Universal Robots PolyScope program: ccc_place_stick.urp

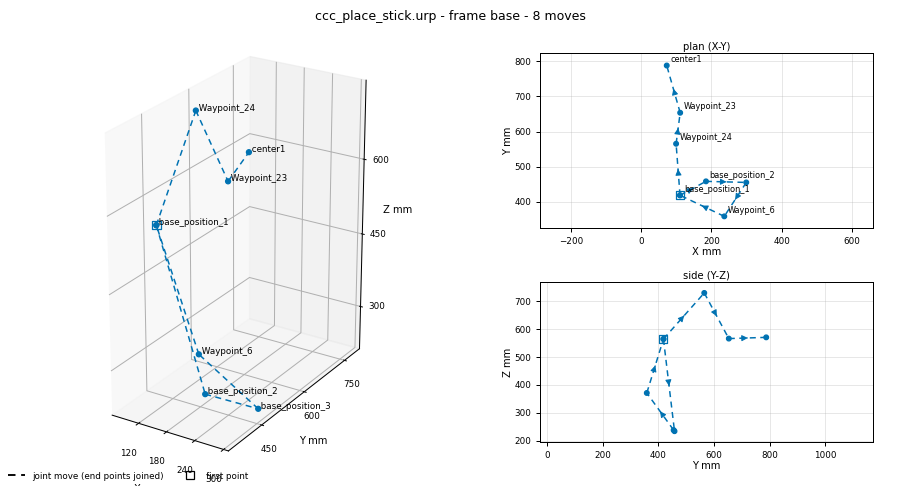
[picture p0: tool path of ccc_place_stick.urp in frame base, 8 of 8 moves have a stored position in this frame; points joined in program order, loops and branches not executed]
Program ccc_place_stick (installation=default directory=/programs/Nicolas_Arteaga/quality createdIn=5.12.4.1101661 lastSavedIn=5.12.4.1101661 robotSerialNumber=20225502378)
Calibrated DH parameters: a=[0.00022, -0.425328, -0.389701, 0.000059, 0.000065, 0]; d=[0.162608, 0.803456, 9.992211, -10.662202, 0.099702, 0.099559]; alpha=[1.570756, 0.001543, 0.004316, 1.570651, -1.570122, 0]; deltaTheta=[0, 0.002917, 0.116094, -0.119008, 0, -0.000001]
Robot Program (runOnlyOnce=true)
  'Takes the first wood stick and places it in the center of the cotton candy machine'
  MoveJ speed 60 deg/s, acceleration 80 deg/s^2 (useActiveTCP=true) feature=Base
    Waypoint base_position_1: TCP in base x=110.873 y=418.875 z=565.206 mm, rx=-1.5602 ry=-0.9891 rz=-1.3624 rad; joints [200.91, -129.117, 99.415, 36.172, 41.428, 90] deg; TCP offset x=0 y=0 z=191.5 mm, rx=0 ry=0 rz=0 rad
    Waypoint base_position_2: TCP in base x=184.715 y=458.614 z=234.006 mm, rx=-1.6866 ry=-0.757 rz=-1.7388 rad; joints [238.232, -104.263, 143.888, -41.533, 99.714, 90.08] deg; TCP offset x=0 y=0 z=191.5 mm, rx=0 ry=0 rz=0 rad
    URCap Gripper Activate (Robotiq_Grippers, Robotiq Inc.) dataModel(ResetAndActivateKey=false)
    URCap Gripper (Robotiq_Grippers, Robotiq Inc.) dataModel(forceInDouble=100.0, speedInDouble=100.0, position=78.0, force=100.0, speed=100.0, positionInDouble=78.0, slaveIds=[9], blocking=true)
    Waypoint base_position_3: TCP in base x=299.306 y=455.502 z=237.992 mm, rx=0.0242 ry=1.587 rz=-0.0069 rad; joints [252.253, -72.527, 107.61, -31.252, 163.421, 274.35] deg; TCP offset x=0 y=0 z=191.5 mm, rx=0 ry=0 rz=0 rad
    stick := GP_int_in[4]
    SuppressedNode
      stick := 10
    Loop While (checkContinuously=false) expression=stick>0
      MoveL speed 250 mm/s, acceleration 1200 mm/s^2 (useActiveTCP=true) feature=Base
        MoveDirectionNode (selectedDirection=ZMinus)
          Until DISTANCE (allowActions=false deceleration=3 distanceNodeType=STOP) Distance=0.016; motionParameters(blendRadius=0)
      stick := stick-1
    MoveL speed 250 mm/s, acceleration 1200 mm/s^2 (useActiveTCP=true) feature=Base
      MoveDirectionNode (selectedDirection=XPlus)
        Until DISTANCE (allowActions=false deceleration=3 distanceNodeType=STOP) Distance=0.022; motionParameters(blendRadius=0)
    URCap Gripper (Robotiq_Grippers, Robotiq Inc.) dataModel(position=100.0, force=0.0, speed=0.0, positionInDouble=100.0, forceInDouble=0.0, speedInDouble=0.0, slaveIds=[9], blocking=true)
    MoveL speed 250 mm/s, acceleration 1200 mm/s^2 (useActiveTCP=true) feature=Base
      MoveDirectionNode (selectedDirection=YMinus)
        Until DISTANCE (allowActions=false deceleration=3 distanceNodeType=STOP) Distance=0.08; motionParameters(blendRadius=0)
    MoveL speed 250 mm/s, acceleration 1200 mm/s^2 (useActiveTCP=true) feature=Base
      MoveDirectionNode (selectedDirection=XMinus)
        Until DISTANCE (allowActions=false deceleration=3 distanceNodeType=STOP) Distance=0.022; motionParameters(blendRadius=0)
    Waypoint Waypoint_6: TCP in base x=236.783 y=359.025 z=371.324 mm, rx=-0.2368 ry=1.6972 rz=-0.2121 rad; joints [256.754, -88.576, 102.057, 18.779, 164.673, 285.268] deg; TCP offset x=0 y=0 z=191.5 mm, rx=0 ry=0 rz=0 rad
    Waypoint Waypoint_28: TCP in base x=110.872 y=418.885 z=565.169 mm, rx=-1.6121 ry=0.3611 rz=-0.2078 rad; joints [200.913, -129.115, 99.418, 36.172, 41.428, 180] deg; TCP offset x=0 y=0 z=191.5 mm, rx=0 ry=0 rz=0 rad
    Waypoint Waypoint_24: TCP in base x=99.712 y=565.5 z=730.734 mm, rx=-1.4619 ry=0.2517 rz=-0.2966 rad; joints [243.031, -99.822, 65.521, 28.761, 83.192, 180] deg; TCP offset x=0 y=0 z=191.5 mm, rx=0 ry=0 rz=0 rad
    Waypoint Waypoint_23: TCP in base x=111.331 y=653.695 z=566.749 mm, rx=-1.7943 ry=0.2693 rz=-0.1351 rad; joints [243.037, -87.632, 65.808, 35.91, 77.265, 180] deg; TCP offset x=0 y=0 z=191.5 mm, rx=0 ry=0 rz=0 rad
    Waypoint center1: TCP in base x=73.065 y=788.054 z=571.181 mm, rx=-1.5688 ry=-0.0203 rz=0.0145 rad; joints [245.634, -75.763, 61.593, 13.883, 64.245, 180.143] deg; TCP offset x=0 y=0 z=191.5 mm, rx=0 ry=0 rz=0 rad
